FUNCTION_BLOCK Test_TExecutionWhenBusy_SetDone_SetsDone EXTENDS T_UnitTestbase
VAR
    Execution : T_Execution;
END_VAR

METHOD Init
SUPER^.Init();

// Setup...
Execution.FB_init(bInitRetains := FALSE,
                  bInCopyCode  := FALSE);
END_METHOD

{attribute 'analysis' := '-33'} // inhibit unused variable warning
METHOD RunTest
// Test...
Execution.Start();
Execution.SetBusy();
Execution.SetDone();

AssertIsTrue(Condition := Execution.Done,
             Message   := 'Execution.Done not true');

AssertIsTrue(Condition := Execution.Ready,
             Message   := 'Execution.Ready not true');

TestCompleted := TRUE;
END_METHOD

END_FUNCTION_BLOCK

(* stored: Version 1.1.0.1, ProductVersion 3.1.4024.12
   POU Test_TExecutionWhenBusy_SetDone_SetsDone: Id {3b0968c7-1b7c-46b9-9efb-9a2380279946}, SpecialFunc None
   Method Init: Id {23cdd901-2538-496b-a1ea-bdb2bbac1a89}
   Method RunTest: Id {f92519b4-385e-4852-a8fe-c1f3edca25b9} *)
